// TwinCAT 3 PLC project PLC2
// ProgramVersion: 3.1.4023.0
// libraries:
//   Tc2_Standard, * (Beckhoff Automation GmbH)
//   Tc2_System, * (Beckhoff Automation GmbH)
//   Tc2_Utilities, * (Beckhoff Automation GmbH)
//   Tc3_Database, * (Beckhoff Automation GmbH)
//   Tc3_EventLogger, * (Beckhoff Automation GmbH)
//   Tc3_IotBase, * (Beckhoff Automation GmbH)
//   Tc3_JsonXml, * (Beckhoff Automation GmbH)
//   Tc3_Module, * (Beckhoff Automation GmbH)
// project tree:
//   DUTs/ aS_DBField.TcDUT
//   GVLs/ GVL.TcGVL
//   / PlcTask.TcTTO
//   POUs/ PostMqtt.TcPOU, ReadDatabase.TcPOU, UpdateSync.TcPOU
// (motion and I/O tree: see PLC project plc1)
// real-time tasks:
//   TASK PlcTask: cycle T#100000us, priority 20, ADS port 350
//   TASK PlcDBTask: cycle T#1ms, priority 21, ADS port 351
//   TASK PlcTask1: cycle T#1ms, priority 22, ADS port 352
// variable links:

CONFIGURATION PLC2
    RESOURCE PLC ON TwinCAT3
        TASK PlcTask(INTERVAL := T#1ms, PRIORITY := 22);
        PROGRAM ReadDatabase WITH PlcTask : ReadDatabase;
        PROGRAM PostMqtt WITH PlcTask : PostMqtt;
        PROGRAM UpdateSync WITH PlcTask : UpdateSync;
    END_RESOURCE
END_CONFIGURATION

// ---- DUTs/aS_DBField.TcDUT
TYPE aS_DBField :
STRUCT
	Id: LINT;
	Sync: BOOL;
	Timestamp: DT;
	FurTemp: REAL;
	FurInper: REAL;
	LphTemp: REAL;
	LphPress: REAL;
	LphInpress: REAL;
	LphInflow: REAL;
	DeaTemp: REAL;
	DeaPress: REAL;
	HphTemp: REAL;
	HphPress: REAL;
	HphInpress: REAL;
	HphInflow: REAL;
	BoiTemp: REAL;
	BoiPress: REAL;
	ConTemp: REAL;
	ConInflow: REAL;
	TurHtemp: REAL;
	TurItemp: REAL;
	TurLtemp: REAL;
	TurHpress: REAL;
	TurIpress: REAL;
	TurLpress: REAL;
	TurSpeed: REAL;
	
	PconMode: BYTE;
	PconRun: BOOL;
	PconVal: REAL;
	PconTime: DINT;
	PconAtime: DINT;
	PconFault: BOOL;
	
	PsupMode: BYTE;
	PsupRun: BOOL;
	PsupVal: REAL;
	PsupTime: DINT;
	PsupAtime: DINT;
	PsupFault: BOOL;
	
	PcirMode: BYTE;
	PcirRun: BOOL;
	PcirVal: REAL;
	PcirTime: DINT;
	PcirAtime: DINT;
	PcirFault: BOOL;
	
	F1Mode: BYTE;
	F1Run: BOOL;
	F1Val: REAL;
	F1Time: DINT;
	F1Atime: DINT;
	F1Fault: BOOL;
	
	F2Mode: BYTE;
	F2Run: BOOL;
	F2Val: REAL;
	F2Time: DINT;
	F2Atime: DINT;
	F2Fault: BOOL;
	
	F3Mode: BYTE;
	F3Run: BOOL;
	F3Val: REAL;
	F3Time: DINT;
	F3Atime: DINT;
	F3Fault: BOOL;
	
	VlphMode: BYTE;
	VlphRun: BOOL;
	VlphVal: REAL;
	VlphTime: DINT;
	VlphAtime: DINT;
	VlphFault: BOOL;
	
	VdeaMode: BYTE;
	VdeaRun: BOOL;
	VdeaVal: REAL;
	VdeaTime: DINT;
	VdeaAtime: DINT;
	VdeaFault: BOOL;
	
	VhphMode: BYTE;
	VhphRun: BOOL;
	VhphVal: REAL;
	VhphTime: DINT;
	VhphAtime: DINT;
	VhphFault: BOOL;
	
	VturMode: BYTE;
	VturRun: BOOL;
	VturVal: REAL;
	VturTime: DINT;
	VturAtime: DINT;
	VturFault: BOOL;
	
	PintMode: BYTE;
	PintRun: BOOL;
	PintVal: REAL;
	PintTime: DINT;
	PintAtime: DINT;
	PintFault: BOOL;
END_STRUCT
END_TYPE

// ---- GVLs/GVL.TcGVL
{attribute 'qualified_only'}
VAR_GLOBAL
	bRemotePosted: BOOL := FALSE;	//Trạng thái đã đẩy lên RemoteDB
	bLocalGot: BOOL:= FALSE;		//Trạng thái đã đọc từ LocalDB
	blocalUpdated: BOOL:= TRUE;	//Trạng thái đã phản hồi LocalDB
	bReExecute: BOOL;
	bMeasure: BOOL;			//Biến để debug
	aReadStruct : aS_DBField;		//Biến lưu dữ liệu tạm từ LocalDB
END_VAR

// ---- POUs/ReadDatabase.TcPOU
PROGRAM ReadDatabase
VAR
	fbSqlDatabase : FB_SQLDatabaseEvt(sNetID := '', tTimeout := T#5S);
	fbSqlCommand : FB_SQLCommandEvt(sNetID := '', tTimeout := T#5S);
	fbSqlResult: FB_SQLResultEvt(sNetID:='', tTimeout := T#5S);
	myDBID: UDINT := 1;			
	sTableName: STRING := 'Data';	
	sCmd: STRING(1000);			

	//Các biến ghi thông báo lỗi	
	tcMessage1 : I_TcMessage;
	tcMessage2 : I_TcMessage;
	tcMessage3 : I_TcMessage;
	tcMessage4 : I_TcMessage;
	
	//Các biến điều khiển
	bFirstScan: BOOL := TRUE;		//Biến báo trạng thái đầu
	bExecute: bool;			//Biến cho phép gửi lệnh SQL
	iId: LINT := 1;			//Biến đếm số lượng bản ghi đã lưu
	bRead: BOOL:= FALSE;		//Biến báo đã đọc được bản ghi
	fbTon: TON;

END_VAR

IF (bFirstScan) THEN
	IF fbSqlDatabase.Connect(myDBID) THEN
		bFirstScan := FALSE;
		IF fbSqlDatabase.bError THEN
			tcMessage1:= fbSqlDatabase.ipTcResult;
			bFirstScan := TRUE;
		END_IF
	END_IF
END_IF

fbTon(IN:= NOT fbTon.Q, PT:= T#1000MS);	
IF fbTon.Q THEN
	bExecute := TRUE;			
END_IF

IF (bExecute OR GVL.bReExecute) AND NOT bFirstScan AND GVL.blocalUpdated THEN
	GVL.bMeasure:= TRUE;	
	CreateSelect();			
		
	IF fbSqlDatabase.CreateCmd(ADR(fbSqlCommand)) THEN	
		IF fbSqlDatabase.bError THEN
			tcMessage2:= fbSqlDatabase.ipTcResult;
		END_IF
	END_IF
		
	IF NOT bRead THEN 	
		IF fbSQLCommand.ExecuteDataReturn(ADR(sCmd), LEN(sCmd), ADR(fbSqlResult)) THEN	
			IF fbSQLCommand.bError THEN
				tcMessage3 := fbSQLCommand.ipTcResult;
			END_IF
			bRead:= TRUE;
		END_IF
	ELSE
		IF fbSqlResult.Read(0, 1, ADR(GVL.aReadStruct), SIZEOF(GVL.aReadStruct), FALSE, TRUE) THEN	
			IF fbSqlResult.bError THEN
				tcMessage4:= fbSqlResult.ipTcResult;
			END_IF
			bRead:= FALSE;	
			bExecute:= FALSE;
			GVL.bReExecute:= FALSE;
	
			IF GVL.aReadStruct.Id <> 0 THEN 
				GVL.blocalUpdated:= FALSE;
				GVL.bLocalGot:= TRUE;
			END_IF
		END_IF
	END_IF
END_IF

ACTION CreateSelect:
sCmd := 'SELECT * FROM ';
sCmd := concat(sCmd, sTableName);
sCmd := concat(sCmd, ' WHERE Sync=0 LIMIT 1');
END_ACTION

END_PROGRAM

// ---- POUs/PostMqtt.TcPOU
PROGRAM PostMqtt
VAR
	fbMqttClient : FB_IotMqttClient;
	bFirstScan : BOOL := TRUE;
	hrErrorOccurred : HRESULT; 
	fbJsonWriter: FB_JsonSaxWriter; 
	
	(* published message *)
	sTopicPub : STRING(255) := 'IPC/ProcessData';
	sPayloadPub : STRING(5000);
	fbTimer : TON;

//	(* received message *)
//	bSubscribed : BOOL;
//	sTopicSub : STRING(255) := 'EK9160/EK-537E06/Stream1/Json/Tx/Data';
//	{attribute 'TcEncoding':='UTF-8'}
//	sTopicRcv : STRING(255);
//	{attribute 'TcEncoding':='UTF-8'}
//	sPayloadSub : STRING(255);
//	fbMessageQueue : FB_IotMqttMessageQueue;
//	fbMessage : FB_IotMqttMessage;

END_VAR

IF bFirstScan THEN
	bFirstScan := FALSE;
	fbMqttClient.sHostName:= '127.0.0.1';
	fbMqttClient.nHostPort:= 8883;
	fbMqttClient.sClientId:= 'mqtt'; 
	fbMqttClient.sTopicPrefix:= ''; 
	fbMqttClient.stTLS.sCA:= 'C:\TwinCAT\3.1\Config\certs\rootCA.pem';
	fbMqttClient.stTLS.bNoServerCertCheck:= TRUE;
	//fbMqttClient.ipMessageQueue := fbMessageQueue;
END_IF

fbMqttClient.Execute(TRUE);
IF fbMqttClient.bError THEN
	hrErrorOccurred := fbMqttClient.hrErrorCode;
END_IF

IF fbMqttClient.bConnected AND GVL.bLocalGot THEN
//	//Subcribe
//	IF NOT bSubscribed THEN
//		bSubscribed := fbMqttClient.Subscribe(sTopic:=sTopicSub, eQoS:=TcIotMqttQos.AtMostOnceDelivery);
//		IF fbMqttClient.bError THEN
//			hrErrorOccurred := fbMqttClient.hrErrorCode;
//		END_IF
//	END_IF
	
	//Publish
	WriteJson();
	fbMqttClient.Publish(	sTopic:= sTopicPub, 
							pPayload:= ADR(sPayloadPub), nPayloadSize:= LEN2(ADR(sPayloadPub))+1, 
							eQoS:= TcIotMqttQos.AtMostOnceDelivery, bRetain:= FALSE, bQueue:= FALSE );
	GVL.bLocalGot := FALSE;
	GVL.bRemotePosted := TRUE;

	IF fbMqttClient.bError THEN
		hrErrorOccurred := fbMqttClient.hrErrorCode;
		GVL.bLocalGot := TRUE;
		GVL.bRemotePosted := FALSE;
	END_IF
END_IF

////Get the subcribe message whenever available
//IF fbMessageQueue.nQueuedMessages > 0 THEN
//	IF fbMessageQueue.Dequeue(fbMessage:=fbMessage) THEN
//		fbMessage.GetTopic(pTopic:=ADR(sTopicRcv), nTopicSize:=SIZEOF(sTopicRcv) );
//		fbMessage.GetPayload(pPayload:=ADR(sPayloadSub), nPayloadSize:=SIZEOF(sPayloadSub), bSetNullTermination:=FALSE);
//	END_IF
//END_IF


//IF GVL.bLocalGot THEN
//	GVL.bLocalGot := FALSE;
//	GVL.bRemotePosted := TRUE;
//END_IF

ACTION WriteJson:
fbJsonWriter.StartObject();
fbJsonWriter.AddKey('Timestamp');
fbJsonWriter.AddDateTime(GVL.aReadStruct.Timestamp);

fbJsonWriter.AddKey('ProcessData');
	fbJsonWriter.StartObject();
	fbJsonWriter.AddKey('FurTemp');
	fbJsonWriter.AddReal(GVL.aReadStruct.FurTemp);
	fbJsonWriter.AddKey('FurInper');
	fbJsonWriter.AddReal(GVL.aReadStruct.FurInper);
	fbJsonWriter.AddKey('LphTemp');
	fbJsonWriter.AddReal(GVL.aReadStruct.LphTemp);
	fbJsonWriter.AddKey('LphPress');
	fbJsonWriter.AddReal(GVL.aReadStruct.LphPress);
	fbJsonWriter.AddKey('LphInpress');
	fbJsonWriter.AddReal(GVL.aReadStruct.LphInpress);
	fbJsonWriter.AddKey('LphInflow');
	fbJsonWriter.AddReal(GVL.aReadStruct.LphInflow);
	fbJsonWriter.AddKey('DeaTemp');
	fbJsonWriter.AddReal(GVL.aReadStruct.DeaTemp);
	fbJsonWriter.AddKey('DeaPress');
	fbJsonWriter.AddReal(GVL.aReadStruct.DeaPress);
	fbJsonWriter.AddKey('HphTemp');
	fbJsonWriter.AddReal(GVL.aReadStruct.HphTemp);
	fbJsonWriter.AddKey('HphPress');
	fbJsonWriter.AddReal(GVL.aReadStruct.HphPress);
	fbJsonWriter.AddKey('HphInpress');
	fbJsonWriter.AddReal(GVL.aReadStruct.HphInpress);
	fbJsonWriter.AddKey('HphInflow');
	fbJsonWriter.AddReal(GVL.aReadStruct.HphInflow);
	fbJsonWriter.AddKey('BoiTemp');
	fbJsonWriter.AddReal(GVL.aReadStruct.BoiTemp);
	fbJsonWriter.AddKey('BoiPress');
	fbJsonWriter.AddReal(GVL.aReadStruct.BoiPress);
	fbJsonWriter.AddKey('ConTemp');
	fbJsonWriter.AddReal(GVL.aReadStruct.ConTemp);
	fbJsonWriter.AddKey('ConInflow');
	fbJsonWriter.AddReal(GVL.aReadStruct.ConInflow);
	fbJsonWriter.AddKey('TurHtemp');
	fbJsonWriter.AddReal(GVL.aReadStruct.TurHtemp);
	fbJsonWriter.AddKey('TurItemp');
	fbJsonWriter.AddReal(GVL.aReadStruct.TurItemp);
	fbJsonWriter.AddKey('TurLtemp');
	fbJsonWriter.AddReal(GVL.aReadStruct.TurLtemp);
	fbJsonWriter.AddKey('TurHpress');
	fbJsonWriter.AddReal(GVL.aReadStruct.TurHpress);
	fbJsonWriter.AddKey('TurIpress');
	fbJsonWriter.AddReal(GVL.aReadStruct.TurIpress);
	fbJsonWriter.AddKey('TurLpress');
	fbJsonWriter.AddReal(GVL.aReadStruct.TurLpress);
	fbJsonWriter.AddKey('TurSpeed');
	fbJsonWriter.AddReal(GVL.aReadStruct.TurSpeed);
	fbJsonWriter.EndObject();
fbJsonWriter.AddKey('ComponentStatus');
	fbJsonWriter.StartObject();
	fbJsonWriter.EndObject();
fbJsonWriter.EndObject();
fbJsonWriter.CopyDocument(sPayloadPub, SIZEOF(sPayloadPub));
fbJsonWriter.ResetDocument();
END_ACTION

END_PROGRAM

// ---- POUs/UpdateSync.TcPOU
PROGRAM UpdateSync
VAR
	fbSqlDatabase : FB_SQLDatabaseEvt(sNetID := '', tTimeout := T#5S);
	fbSqlCommand : FB_SQLCommandEvt(sNetID := '', tTimeout := T#5S);
	myDBID: UDINT := 1;		
	sTableName: STRING := 'Data';	
	sCmd: STRING(1000);			
		
	tcMessage1 : I_TcMessage;
	tcMessage2 : I_TcMessage;

	bFirstScan: BOOL := TRUE;

END_VAR

IF (bFirstScan) THEN
	IF fbSqlDatabase.Connect(myDBID) THEN
		bFirstScan := FALSE;
		IF fbSqlDatabase.bError THEN
			tcMessage1:= fbSqlDatabase.ipTcResult;
			bFirstScan := TRUE;
		END_IF
	END_IF
END_IF

IF GVL.bRemotePosted THEN
	CreateUpdate();		
		
	IF fbSqlDatabase.CreateCmd(ADR(fbSqlCommand)) THEN  
		IF fbSqlDatabase.bError THEN
			tcMessage1:= fbSqlDatabase.ipTcResult;
		END_IF
	END_IF
		
	IF fbSQLCommand.Execute(ADR(sCmd), LEN(sCmd)) THEN	
		IF fbSQLCommand.bError THEN
			tcMessage2 := fbSQLCommand.ipTcResult;
		END_IF
		
		GVL.bRemotePosted := FALSE;
		gvl.blocalUpdated := TRUE;
		GVL.bReExecute := TRUE;
		GVL.bMeasure := FALSE;
	END_IF
END_IF

ACTION CreateUpdate:
sCmd := 'UPDATE ';
sCmd := concat(sCmd, sTableName);
sCmd := concat(sCmd, ' SET Sync=');
sCmd := concat(sCmd, BOOL_TO_STRING(TRUE));
sCmd := concat(sCmd, ' WHERE Id=');
sCmd := concat(sCmd, LINT_TO_STRING(GVL.aReadStruct.Id));
END_ACTION

END_PROGRAM
